// TIA Portal V18 export
DATA_BLOCK "Emergency_DB"   // DB22
{ S7_Optimized_Access := 'FALSE' }
VERSION : 0.1
// stored: AutoNumber true, IsOnlyStoredInLoadMemory false, IsWriteProtectedInAS false
   VAR
      Emergency_1 : Bool;
      Emergency_2 : Bool;
      Emergency_3 : Bool;
      Emergency_4 : Bool;
      Emergency_5 : Bool;
      Emergency_6 : Bool;
      Emergency_7 : Bool;
      Emergency_8 : Bool;
      Emergency_9 : Bool;
      Emergency_10 : Bool;
      Emergency_11 : Bool;
      Emergency_12 : Bool;
      Emergency_13 : Bool;
      Emergency_14 : Bool;
      Emergency_15 : Bool;
      Emergency_16 : Bool;
   END_VAR
BEGIN
END_DATA_BLOCK
